(* IEC 61131-3 sources: SHU_NSTV/src/lib/PumpLib, 6 files *)

(* ---- IPumpVFD_Control.st ---- *)
INTERFACE IPumpVFD_Control EXTENDS BasicControl

    METHOD Set_Power_VFD
    VAR_INPUT
        x : BOOL;
    END_VAR

    PROPERTY PowerVFD : BOOL
    (* 	from: BasicControl
    * 	Чтобы получить выходной сигнал из функционального блока, требуется вызвать свойство Power.
    *	Значение Power можно присовить, например, на питание контактора исполнительного механизма.	-	-	-	-	-	-	-	-	: PU1_KM_cmdOn := PU1.Power;
    *	Чтобы получить сигнал работы от механизма, требуется записать сигнал механизма в свойство Power	-	-	-	-	-	-	-	: PU1.Power := PU1_KM_On;
    *																																^
    *	Важно: Логика функционального блока подразумевает, что свойство Power будет присвоено на питание контактора,				^
    *	а сигнал работы исполнительного механизма (статус: включён) будет присовен внутрь свойства Power. Как показано на примере выше.
    *)

(* ---- IPumpVFD_ControlCommands.st ---- *)
INTERFACE IPumpVFD_ControlCommands EXTENDS BasicControlCommands

    METHOD Start_VFD
    VAR_INPUT
        access : BOOL;
        device : IPumpVFD_Control;
    END_VAR

    METHOD Stop_VFD
    VAR_INPUT
        access: BOOL;
        device : IPumpVFD_Control;
    END_VAR

    METHOD SwitchToStart
    VAR_INPUT
        access : BOOL;
        device : IPumpVFD_Control;
    END_VAR
    METHOD SwitchToVFD
    VAR_INPUT
        access : BOOL;
        device : IPumpVFD_Control;
    END_VAR

(* ---- Pump_Control.st ---- *)
FUNCTION_BLOCK Pump_Control IMPLEMENTS BasicControlCommands
VAR_INPUT
END_VAR
VAR_OUTPUT
END_VAR
VAR
	ConditionStart : BOOL;						// Условие на запуск
	ConditionStop : BOOL; 						// Условие на стоп.
END_VAR

METHOD Start
    VAR_INPUT
        access : BOOL;							// Доступ к запуску
        device : BasicControl;				        // Устройство управления насосом
    END_VAR

    IF access AND ConditionStart THEN
        device.Set_Power(TRUE);					// Запускаем насос
    END_IF;
END_METHOD

METHOD Stop
    VAR_INPUT
        access: BOOL;							// Доступ к остановке
        device : BasicControl;				        // Устройство управления насосом
    END_VAR

    IF access AND ConditionStop THEN
        device.Set_Power(FALSE);				// Останавливаем насос
    END_IF;
END_METHOD

PROPERTY AccessToStart : BOOL
    SET
        ConditionStart := AccessToStart;
    END_GET
END_PROPERTY

PROPERTY AccessToStop : BOOL
    SET
        ConditionStop := AccessToStop;
    END_GET
END_PROPERTY
END_FUNCTION_BLOCK

(* ---- Pump_Control_VFD.st ---- *)
FUNCTION_BLOCK Pump_Control_VFD EXTENDS Pump_Control IMPLEMENTS IPumpVFD_ControlCommands
VAR_INPUT
END_VAR
VAR_OUTPUT
END_VAR
VAR
	ConditionStartVFD : BOOL;								// Переменная услвоия старта насоса от ЧРП
	ConditionSwitchToStart, ConditionSwitchToVFD : BOOL;	// Условия перехода насоса на ЧРП и обычный старт
END_VAR

METHOD Start_VFD
    VAR_INPUT
        access : BOOL;										// Доступ к функциональному блоку
        device : IPumpVFD_Control;							// Устройство управления насосом от ЧРП
    END_VAR

    IF access AND ConditionStartVFD THEN
        device.Set_Power_VFD(TRUE);
    END_IF;
END_METHOD

METHOD Stop_VFD
    VAR_INPUT
        access: BOOL;										// Доступ к функциональному блоку
        device : IPumpVFD_Control;							// Устройство управления насосом от ЧРП
    END_VAR

    IF access AND ConditionStop THEN
        device.Set_Power_VFD(FALSE);
    END_IF;
END_METHOD

METHOD SwitchToStart
    VAR_INPUT
        access : BOOL;										// Доступ к функциональному блоку
        device : IPumpVFD_Control;							// Устройство управления насосом от ЧРП
    END_VAR

    IF access AND ConditionSwitchToStart THEN
        device.Set_Power_VFD(FALSE);
        device.Set_Power(TRUE);
    END_IF;
END_METHOD

METHOD SwitchToVFD
    VAR_INPUT
        access : BOOL;										// Доступ к функциональному блоку
        device : IPumpVFD_Control;							// Устройство управления насосом от ЧРП
    END_VAR

    IF access AND ConditionSwitchToVFD THEN
        device.Set_Power(FALSE);
        device.Set_Power_VFD(TRUE);
    END_IF;
END_METHOD

PROPERTY AccessToStartVFD : BOOL
    SET
        ConditionStartVFD := AccessToStartVFD;
    END_SET
END_PROPERTY

PROPERTY AccessToSwitchToStart : BOOL
    SET
        ConditionSwitchToStart := AccessToSwitchToStart;
    END_SET
END_PROPERTY

PROPERTY AccessToSwitchToVFD : BOOL
    SET
        ConditionSwitchToVFD := AccessToSwitchToVFD;
    END_SET
END_PROPERTY
END_FUNCTION_BLOCK

(* ---- Pump_VFD.st ---- *)
FUNCTION_BLOCK Pump_VFD EXTENDS PumpBasic IMPLEMENTS IPumpVFD_Control
VAR_INPUT
END_VAR
VAR_OUTPUT
END_VAR
VAR
	qxPowerVFD : BOOL;			// Выходной сигнал: 	Питание от ЧРП
END_VAR

METHOD Set_Power_VFD
    VAR_INPUT
        x : BOOL;				// Входной сигнал: 	Питание от ЧРП
    END_VAR
    qxPowerVFD := x;			// Присваиваем значение входного сигнала питания к выходному сигналу
END_METHOD
PROPERTY PowerVFD : BOOL
    GET
        PowerVFD := qxPowerVFD;	// Возвращаем значение выходного сигнала питания от ЧРП
    END_GET
END_PROPERTY
END_FUNCTION_BLOCK

(* ---- PumpBasic.st ---- *)
FUNCTION_BLOCK PumpBasic IMPLEMENTS BasicControl
VAR_INPUT
END_VAR
VAR_OUTPUT
END_VAR
VAR
	qxPower : BOOL;			// Выход сигнала питания
END_VAR

METHOD Set_Power
    VAR_INPUT
        x : BOOL;				// Вход сигнала питания
    END_VAR
    qxPower := x;				// Присваиваем значение входного сигнала питания к выходному сигналу
END_METHOD

PROPERTY Power : BOOL
    GET
        Power := qxPower;	// Возвращаем значение выходного сигнала питания
    END_GET
END_PROPERTY
END_FUNCTION_BLOCK
